TYPE ST_DeviceRecipe :
STRUCT
	Ateq 		: ARRAY[0..GVL_AteqConfig.nMaxDeviceCount] OF ST_AteqRecipe;
	ValveBank	: ARRAY[0..GVL_ValveBankConfig.nMaxDeviceCount] OF ST_RecipeTypeValveBank;
END_STRUCT
END_TYPE

(* stored: Version 1.1.0.1
   DUT ST_DeviceRecipe: Id {a894167e-fbab-0500-0e58-42976805dbb1} *)
